FUNCTION_BLOCK FB_TCPClient

VAR_INPUT
	sRemoteHost: T_IPv4Addr;
	nRemotePort: UDINT;
	sSendData: ARRAY[0..1023] OF BYTE;;	
	bStartCommunication: BOOL;
	tCycleTimeSend: TIME;
	bSendTrigger : BOOL;
END_VAR

VAR_OUTPUT
	bConnected: BOOL;
	sReceivedData: ARRAY[0..1023] OF BYTE;
	nErrorID: UDINT;
	bError: BOOL;
	bBusy: BOOL;
END_VAR

VAR
	iState: INT;
	fbSocketConnect: FB_SocketConnect;
	fbSocketSend: FB_SocketSend;
	deserialize: deserialize;
	fbSocketClose: FB_SocketClose;
	fbSocketReceive: FB_SocketReceive;
	hSocket: T_HSOCKET;

	fbTimer: TON;
	nRecBytes: UDINT;
	bExecuteSocketSend: BOOL;
	RTrig: R_TRIG;
	buffer : UDINT;
END_VAR

CASE iState OF
	0:	// Init State
		fbSocketConnect(bExecute := FALSE); 
		fbSocketSend(bExecute := FALSE); 
		fbSocketReceive(bExecute := FALSE);
		fbSocketClose(bExecute := FALSE); 
		bConnected := FALSE; 
		bBusy := FALSE;
		IF bStartCommunication = TRUE THEN									// Start communication manually 
			iState := iState + 10;
			bBusy := TRUE;
			bError := FALSE;
		END_IF
	
	10:	// Connect Server
		fbSocketConnect(													// Open connection to server
			sSrvNetId:= '', 
			sRemoteHost:= sRemoteHost, 
			nRemotePort:= nRemotePort, 
			bExecute:= TRUE, 
			tTimeout:= T#4S, 
			bBusy=> , 
			bError=> bError, 
			nErrId=> nErrorID, 
			hSocket=> hSocket);
	
		IF hSocket.handle <> 0 AND NOT (fbSocketConnect.bBusy) THEN			// Handle is created
			bConnected := TRUE; 
			iState :=iState + 5;
		ELSIF bError THEN
			iState := 0; 	
		END_IF
		
		
	15:																		// StartCommunication
		IF (tCycleTimeSend <> T#0MS) THEN									// Send data cyclically
			fbTimer(IN:= NOT fbTimer.Q, PT:= tCycleTimeSend, Q=> , ET=> );		
		END_IF
		RTrig(CLK:= bSendTrigger, Q=> );									// SendData on manuel trigger
		
		fbSocketSend(														// Send Data
			sSrvNetId:= '', 
			hSocket:= hSocket, 
			cbLen:= SIZEOF(sSendData), 
			pSrc:= ADR(sSendData), 
			bExecute:= (fbTimer.Q OR RTrig.Q), 
			tTimeout:= T#2S, 
			bError=> bError, 
			nErrId=> nErrorID, 
			nErrId=> );
	
		fbSocketReceive(													// ReceiveData
			sSrvNetId:= '', 
			hSocket:= hSocket, 
			cbLen:= SIZEOF(sReceivedData), 
			pDest:= ADR(sReceivedData), 
			bExecute:= true, 
			tTimeout:= T#3S, 
			bBusy=> , 
			bError=> bError, 
			nErrId=> nErrorID, 
			nRecBytes=> nRecBytes);
	
		IF NOT fbSocketReceive.bBusy THEN									// Check cyclically for new data
			fbSocketReceive(bExecute := FALSE);
		END_IF						
		IF NOT bStartCommunication OR bError THEN							// Close connection in case of error or manual communication stop
			iState := 20;
		END_IF
	20: 
		fbSocketClose(														// Close connection
			sSrvNetId:= '', 
			hSocket:= hSocket, 
			bExecute:= TRUE, 
			tTimeout:= T#4S, 
			bBusy=> , 
			bError=> bError, 
			nErrId=> nErrorID );
		IF NOT fbSocketClose.bBusy THEN
			iState :=0;		
		END_IF
END_CASE

END_FUNCTION_BLOCK

(* stored: Version 1.1.0.1, ProductVersion 3.1.4024.13
   POU FB_TCPClient: Id {aee5fad7-6181-4fcb-97d6-7d2836584029}, SpecialFunc None *)
